// TIA Portal V20 export
FUNCTION_BLOCK "FB_Lad"   // FB5, LAD
{ S7_Optimized_Access := 'TRUE' }
   VAR_INPUT
      Start : Bool;
   END_VAR
   VAR_OUTPUT
      Done : Bool;   // sequence finished
   END_VAR
   VAR
      Cfg : Struct
         Limit : Int := 10;
      END_STRUCT;
      Hist : Array[0..3] of Real;
      Motor : "ST_Motor";
   END_VAR
BEGIN
END_FUNCTION_BLOCK
